TYPE ST_TCSubModuleEPT :
STRUCT
	TCSite: ARRAY [1..(.NO_OF_TC_SITE)] OF ST_TCUEPT;
END_STRUCT
END_TYPE

(* stored: Version 1.1.0.1, ProductVersion 3.1.4022.12
   DUT ST_TCSubModuleEPT: Id {6a76e2d4-a735-4cae-b035-a35b2854a0b6} *)
